FUNCTION_BLOCK FB_AnalogIn
VAR_INPUT 
	iMaxInCH : INT;
END_VAR
VAR_OUTPUT
END_VAR
VAR
	//AnalogIn	: ARRAY [1..GVL_AnalogInputs.iAIChannelCount] OF AI_config;
	iIndex 		: INT;
	iMax		: INT;
END_VAR

IF iMaxInCH > GVL_AnalogInputs.iAIChannelCount THEN
	iMax := GVL_AnalogInputs.iAIChannelCount;
ELSE
	iMax := iMaxInCH;
END_IF

FOR iIndex :=1 TO iMax BY 1 DO
	(*IF GVL_AnalogInputs.iAinChannel[iIndex]>0 THEN*)
	GVL_AnalogInputs.hmi_config[iIndex].rRawUnits:= Count_to_MeasureUnits
		(
		iValue_in	:=	GVL_AnalogInputs.hmi_config[iIndex].iRawCount,
		iHigh		:=	20,
		iLow		:= 	4
		);
		
	GVL_AnalogInputs.hmi_config[iIndex].rEngUnit:= MeasureUnit_to_EngUnits
		(	
		rValue:= GVL_AnalogInputs.hmi_config[iIndex].rRawUnits,
		rSlope:= GVL_AnalogInputs.hmi_config[iIndex].slope,
		rOffset:=GVL_AnalogInputs.hmi_config[iIndex].offset
		);
		
END_FOR

END_FUNCTION_BLOCK

(* stored: Version 1.1.0.1, ProductVersion 3.1.4024.12
   POU FB_AnalogIn: Id {b9d98d80-fd6d-4389-9ffe-23aaf7609279}, SpecialFunc None *)
